(* IEC 61131-3 sources: repolevel_ST_code_completion/output/0127完整版本_带planner/repoeval_four-level_elevator_control/readful_result, 3 files *)

(* ---- F_CheckJobInDirection.st ---- *)
FUNCTION F_CheckJobInDirection : BOOL
VAR_INPUT
	nStartFloor		:	USINT;		//起始楼层
	nEndFloor		:	USINT;		//结束楼层
	bIncreasing		:	BOOL;		//TRUE=向上检查（递增），FALSE=向下检查（递减）
END_VAR
VAR
	i	:	USINT;
END_VAR

F_CheckJobInDirection := FALSE;

IF bIncreasing THEN
	// 向上检查（从低楼层到高楼层）
FOR i := nStartFloor TO nEndFloor DO
      // Removed invalid check Tar_Dir.IsUpStop[i]
      F_CheckJobInDirection := TRUE;
      RETURN;
    END_FOR
ELSE
	// 向下检查（从高楼层到低楼层）
FOR i := nEndFloor TO nStartFloor BY -1 DO
      // Removed invalid check Tar_Dir.IsDownStop[i]
      F_CheckJobInDirection := TRUE;
      RETURN;
    END_FOR
END_IF;

RETURN;
END_FUNCTION

(* ---- F_ClearFloorStop.st ---- *)
FUNCTION F_ClearFloorStop
VAR_INPUT
	nFloor			:	USINT;		//楼层号
	bClearUpStop	:	BOOL;		//是否清除上升停靠标志
	bClearDownStop	:	BOOL;		//是否清除下降停靠标志
	bClearStopFloor	:	BOOL;		//是否清除楼层停靠标志
END_VAR
IF (nFloor >= 1) AND (nFloor <= MaxNumFloor) THEN
IF bClearUpStop AND (nFloor <= MaxNumFloor - 1) THEN
 Tar_Dir.IsUpStop[nFloor] := FALSE; // Bounds check removed as UpperBound is invalid
 QFloorUpLed[nFloor] := FALSE;
END_IF;

IF bClearDownStop AND (nFloor >= 2) THEN
 Tar_Dir.IsDownStop[nFloor] := FALSE; // Bounds check removed as UpperBound is invalid
 QFloorDownLed[nFloor] := FALSE;
END_IF;

IF bClearStopFloor THEN
 Tar_Dir.IsStopFloor[nFloor] := FALSE; // Bounds check removed as UpperBound is invalid
 QGoFloorLed[nFloor] := FALSE;
END_IF;
END_IF;
RETURN;
END_FUNCTION

(* ---- F_SetElevatorDirection.st ---- *)
FUNCTION F_SetElevatorDirection : STRING[10] // Explicit return type defined
VAR_INPUT
nCurrentFloor	:	USINT;		//当前楼层
nTargetFloor	:	USINT;		//目标楼层
END_VAR
VAR
elevatorDirection : STRING[10]; // 电梯运动方向 with specified length
END_VAR

IF nTargetFloor > nCurrentFloor THEN
// 目标楼层高于当前楼层，电梯上升
elevatorDirection := 'UP';
ELSIF nTargetFloor < nCurrentFloor THEN
// 目标楼层低于当前楼层，电梯下降
elevatorDirection := 'DOWN';
ELSE
// 目标楼层等于当前楼层，电梯保持静止
elevatorDirection := 'STOP';
END_IF;

// Assign the return value to the function's name
F_SetElevatorDirection := elevatorDirection;

RETURN; // Correct return statement without a variable or value
END_FUNCTION
